// TIA Portal V19 export
TYPE "UDT_MOTOR"
   STRUCT
      cmd : Struct   // Commands
         auto : Bool := false;
         man : Bool := false;
         start : Bool := false;
         stop : Bool := false;
      END_STRUCT;
      ind : Struct
         auto : Bool := false;
         man : Bool := false;
         start : Bool := false;
         stop : Bool := false;
      END_STRUCT;
      sim : Struct   // Simulation
         fb { S7_SetPoint := 'True'} : Bool := false;   // Feedback simulation
         ctrl { S7_SetPoint := 'True'} : Bool := false;   // Control simulation
      END_STRUCT;
      faults : Struct   // Faults
         ftr { S7_SetPoint := 'True'} : "UDT_ALARMACKN";   // Fail to run
         fts { S7_SetPoint := 'True'} : "UDT_ALARMACKN";   // Fail to stop
         mcb { S7_SetPoint := 'True'} : "UDT_ALARMACKN";   // MCB failure
         ctrl { S7_SetPoint := 'True'} : "UDT_ALARMACKN";   // CTRL failure
         vfd { S7_SetPoint := 'True'} : "UDT_ALARMACKN";   // VFD failure
         il { S7_SetPoint := 'True'} : "UDT_ALARMACKN";   // Interlock violation
         fpreset : Bool := false;   // Faceplate reset for individual treatment
      END_STRUCT;
      pid : Struct   // PID
         mode { S7_SetPoint := 'True'} : Bool := false;   // Auto=0, Man=1
         action { S7_SetPoint := 'True'} : Bool := false;   // Reverse=0, Forward=1
         spsource : Bool := false;   // 0=internal setpoint, 1=external setpoint
         followup : Bool := false;   // 0=motor control from PID, 1=motor setpoint directly from program
         cmdrst : Bool := false;   // Controller reset command
         pidrun : Bool := false;   // Controller is running
         P { S7_SetPoint := 'True'} : Real := 0.0;   // Proportional gain
         I { S7_SetPoint := 'True'} : DInt := 0;   // Integral action
         D { S7_SetPoint := 'True'} : DInt := 0;   // Derivative action
         SP { S7_SetPoint := 'True'} : Real := 0.0;   // Setpoint
         PV : Real := 0.0;   // Peripheral value (Reference value for PID)
         OFFVAL { S7_SetPoint := 'True'} : Real := 0.0;   // Value loaded to OP when the actuator is stopped
         LMN : Real := 0.0;   // Output of the PID controller
         OP { S7_SetPoint := 'True'} : Real := 0.0;   // Final output to the element
         L { S7_SetPoint := 'True'} : Real := 0.0;   // Lower value
         H { S7_SetPoint := 'True'} : Real := 0.0;   // Higher value
         EXT_SP : Real := 0.0;   // External setpoint
         FUP : Real := 0.0;   // Follow up value
         ITLVAL { S7_SetPoint := 'True'} : Real := 0.0;   // Controller initialization value
         pvunit { S7_SetPoint := 'True'} : WString := WSTRING#'';   // Unit
         outunit { S7_SetPoint := 'True'} : WString := WSTRING#'';   // Output Unit
         init : Struct   // Controller initialization routine
            req : Bool := false;   // An initialization routine is required
            dur { S7_SetPoint := 'True'} : Real := 0.0;   // Initialization duration
            delay : "UDT_DELAYON";   // UDT_DELAYONOFF
         END_STRUCT;
      END_STRUCT;
      unscale : Struct   // Scale output
         in : Real := 0.0;   // Value to be unscaled
         inhigh { S7_SetPoint := 'True'} : Real := 0.0;   // High limit of scale process (input value)
         inlow { S7_SetPoint := 'True'} : Real := 0.0;   // Low limit of scale process (input value)
         outhigh { S7_SetPoint := 'True'} : Real := 0.0;   // High limit of scale process (output value)
         outlow { S7_SetPoint := 'True'} : Real := 0.0;   // Low limit of scale process (output value)
         output : Real := 0.0;   // Unscaled value (only linear and span > 0)
         set : Bool := false;   // The scaling function is set
      END_STRUCT;
      arh : Struct   // Working hours & maintenance timer
         checkafter { S7_SetPoint := 'True'} : DInt := 0;   // Check motor after this SP of working hours
         lastmaint : DInt := 0;   // Last maintenance
         difference : DInt := 0;   // Actual - Last maintenance
         actual : DInt := 0;   // Actual working time (h)
         seconds : DInt := 0;   // seconds counter
         hour : Bool := false;   // 1 hour completed
         resetarh : Bool := false;   // Reset total timer
         enable : Bool := false;   // Enable maintenance
         maintenance : Bool := false;   // Maintenance required
         completed : Bool := false;   // Maintenance completed
      END_STRUCT;
      status : Struct   // Status
         vfb : Bool := false;   // Virtual feedback
         vctrl : Bool := false;   // Virtual control
         ilstart : Bool := false;   // Motor is allowed to start
         fault : Bool := false;   // General fault (generated from the others)
         maint : Bool := false;   // Maintenance required
         icon : Int := 0;
      END_STRUCT;
      delay { S7_SetPoint := 'True'} : "UDT_DELAYONOFF";   // Activation delay on/off
      out : Struct   // Output
         manrun : Bool := false;   // Manual run
         run : Bool := false;   // Command to run
         ref : Int := 0;   // Unscaled value to be loaded to the next channel (vfd, aq, etc)
      END_STRUCT;
   END_STRUCT;
END_TYPE
